(* PLC project HydMotion Functions library, Porcheson AuxBAse Framework 0.0 *)
(* stored: creationDateTime 2023-02-10T00:00:00, modificationDateTime 2026-02-10T00:00:00 *)

TYPE HDY_AxisMotion : STRUCT
  SEGMENTTAG : USINT;
  PLANNER : USINT;
  MODE : USINT;
  ENDCONDITION : USINT;
  DIRECTION : USINT;
  SETPOSITION : REAL;
  SETVELOCITY : REAL;  (* 仅在速度/流量控制模式下使用，表示目标速度； *)
  SETFLOW : REAL;  (* 仅在速度/流量控制模式下使用，表示目标流量；在位置控制模式下忽略 *)
  SETPRESSURE : REAL;
  ACCELERATION : REAL;
  DECELERATION : REAL;
  DURATION : REAL;
  PRESSURERAMPRATE : REAL;
  ACTPOSITION : REAL;
  ACTVELOCITY : REAL;
  ACTFLOW : REAL;
  ACTPRESSURE : REAL;
  TIMESTAMP : REAL;
END_STRUCT;
END_TYPE

FUNCTION_BLOCK HDY_MoveProfile
  VAR_INPUT
    EXECUTE : BOOL;
    MOTION : HDY_AxisMotion;
    AXISID : SINT;
    BUFFERMODE : INT;
  END_VAR
  VAR_OUTPUT
    ACTIVE : BOOL;
    BUSY : BOOL;
    DONE : BOOL;
    ERROR : BOOL;
    ERRORID : WORD;
  END_VAR
  VAR
    Execute0 : BOOL;
    Done0 : BOOL;
    Active0 : BOOL;
    _PENDING : BOOL;
    _EXEC_ID : WORD;
  END_VAR

 {{ extern void __mcl_cmd_MoveProfile(HDY_MOVEPROFILE *data__);	__mcl_cmd_MoveProfile(data__);	 }}			
END_FUNCTION_BLOCK

FUNCTION_BLOCK HDY_LoadProfile
  VAR_INPUT
    EXECUTE : BOOL;
    AXISID : SINT;
    MOTION : HDY_AxisMotion;
  END_VAR
  VAR_OUTPUT
    BUSY : BOOL;
    DONE : BOOL;
    ERROR : BOOL;
    ERRORID : WORD;
  END_VAR
  VAR
    Execute0 : BOOL;
    Done0 : BOOL;
  END_VAR

						{{ extern void __mcl_cmd_LoadProfile(HDY_LOADPROFILE *data__);	__mcl_cmd_LoadProfile(data__);	 }}	
					
END_FUNCTION_BLOCK

FUNCTION_BLOCK HDY_Stop
  VAR_INPUT
    EXECUTE : BOOL;
    AXISID : SINT;
    DECELERATION : REAL;
  END_VAR
  VAR_OUTPUT
    BUSY : BOOL;
    DONE : BOOL;
    COMMANDABORTED : BOOL;
    ERROR : BOOL;
    ERRORID : WORD;
  END_VAR
  VAR
    Execute0 : BOOL;
    Done0 : BOOL;
    Active0 : BOOL;
    _PENDING : BOOL;
  END_VAR

						{{ extern void __mcl_cmd_Stop(HDY_STOP *data__);	__mcl_cmd_Stop(data__);	 }}	
					
END_FUNCTION_BLOCK

(* This Function Block commands a controlled motion to a specified absolute position. *)
FUNCTION_BLOCK HDY_MoveAbsolute
  VAR_INPUT
    EXECUTE : BOOL;
    AXISID : SINT;
    ContinuousUpdate : BOOL;
    POSITION : REAL;
    VELOCITY : REAL;
    ACCELERATION : REAL;
    DECELERATION : REAL;
    JERK : REAL;
    DIRECTION : SINT;
    BUFFERMODE : INT;
  END_VAR
  VAR_OUTPUT
    DONE : BOOL;
    BUSY : BOOL;
    ACTIVE : BOOL;
    COMMANDABORTED : BOOL;
    ERROR : BOOL;
    ERRORID : WORD;
  END_VAR
  VAR
    EXECUTE0 : BOOL;
    DONE0 : BOOL;
    ACTIVE0 : BOOL;
    _PENDING : BOOL;
    _EXEC_ID : WORD;
  END_VAR

						{{ extern void __mcl_cmd_MoveAbsolute(HDY_MOVEABSOLUTE*); __mcl_cmd_MoveAbsolute(data__); }}	
					
END_FUNCTION_BLOCK

(* This Function Block commands a never ending controlled motion at a specified velocity. *)
FUNCTION_BLOCK HDY_MoveVelocity
  VAR_INPUT
    EXECUTE : BOOL;
    AXISID : SINT;
    CONTINUOUSUPDATE : BOOL;
    VELOCITY : REAL;
    ACCELERATION : REAL;
    DECELERATION : REAL;
    JERK : REAL;
    DIRECTION : SINT;
    BUFFERMODE : INT;
  END_VAR
  VAR_OUTPUT
    INVELOCITY : BOOL;
    BUSY : BOOL;
    ACTIVE : BOOL;
    COMMANDABORTED : BOOL;
    ERROR : BOOL;
    ERRORID : WORD;
  END_VAR
  VAR
    EXECUTE0 : BOOL;
    INVELOCITY0 : BOOL;
    ACTIVE0 : BOOL;
    _PENDING : BOOL;
    _EXEC_ID : WORD;
  END_VAR

{{ extern void __mcl_cmd_MoveVelocity(HDY_MOVEVELOCITY*); __mcl_cmd_MoveVelocity(data__); }} 
END_FUNCTION_BLOCK

(* This Function Block makes the transition from the state ‘ErrorStop’ to ‘Disabled’ by resetting all internal axis-related errors *)
FUNCTION_BLOCK HDY_Reset
  VAR_INPUT
    EXECUTE : BOOL;
    AXISID : SINT;
  END_VAR
  VAR_OUTPUT
    DONE : BOOL;
    BUSY : BOOL;
    ERROR : BOOL;
    ERRORID : WORD;
  END_VAR
  VAR
    EXECUTE0 : BOOL;
    DONE0 : BOOL;
  END_VAR

{{ extern void __mcl_cmd_Reset(HDY_RESET*); __mcl_cmd_Reset(data__); }} 
END_FUNCTION_BLOCK

(* This Function Block commands pressure closed control. *)
FUNCTION_BLOCK HDY_PressureHandle
  VAR_INPUT
    EXECUTE : BOOL;
    AXISID : SINT;
    PRESSURE : REAL;
    PRESSURERAMPRATE : REAL;
    DURATION : REAL;
    BUFFERMODE : INT;
  END_VAR
  VAR_OUTPUT
    INPRESSURE : BOOL;
    BUSY : BOOL;
    ACTIVE : BOOL;
    COMMANDABORTED : BOOL;
    ERROR : BOOL;
    ERRORID : WORD;
  END_VAR
  VAR
    EXECUTE0 : BOOL;
    INPRESSURE0 : BOOL;
    ACTIVE0 : BOOL;
    _PENDING : BOOL;
    _EXEC_ID : WORD;
  END_VAR

{{ extern void __mcl_cmd_PressureHandle(HDY_PRESSUREHANDLE*); __mcl_cmd_PressureHandle(data__); }} 
END_FUNCTION_BLOCK

(* This allocates a simulation Axis, for testing.One axis per instanciated FB. *)
FUNCTION_BLOCK HDY_CreateMotion
  VAR_INPUT
    USE_RECIPE : BOOL := 0;
    FLOW_TO_PUMPSPEED : REAL := 20.0;
    PUMPSPEED_LIMIT : REAL := 1800.0;
    USE_SIMULATION : BOOL := 0;
  END_VAR
  VAR_OUTPUT
    AXISID : SINT;
    BUSY : BOOL;
    DONE : BOOL;
    ERROR : BOOL;
    ERRORID : WORD;
  END_VAR
  VAR
    DONE0 : BOOL;
  END_VAR

						{{ extern void __mcl_cmd_CreateMotion(HDY_CREATEMOTION*); __mcl_cmd_CreateMotion(data__); }} 
					
END_FUNCTION_BLOCK

(* set feedback to motion. *)
FUNCTION_BLOCK HDY_SetAxisFeedback
  VAR_INPUT
    ENABLE : BOOL;
    AXISID : SINT;
    ACT_POSITION : REAL;
    ACT_VELOCITY : REAL;
    ACT_FLOW : REAL;
    ACT_PRESSURE : REAL;
    TIMESTAMP : REAL;
  END_VAR
  VAR_OUTPUT
    BUSY : BOOL;
    DONE : BOOL;
    ERROR : BOOL;
    ERRORID : WORD;
  END_VAR
  VAR
    DONE0 : BOOL;
  END_VAR

						{{ extern void __mcl_cmd_SetAxisFeedback(HDY_SETAXISFEEDBACK*); __mcl_cmd_SetAxisFeedback(data__); }} 
					
END_FUNCTION_BLOCK

(* get only one pump speed command from motion. *)
FUNCTION_BLOCK HDY_GetPumpRequest
  VAR_INPUT
    ENABLE : BOOL;
    STRATEGY : SINT;
  END_VAR
  VAR_OUTPUT
    PUMPSPEED : REAL;
    BUSY : BOOL;
    DONE : BOOL;
    ERROR : BOOL;
    ERRORID : WORD;
  END_VAR
  VAR
    DONE0 : BOOL;
  END_VAR

						{{ extern void __mcl_cmd_GetPumpRequest(HDY_GETPUMPREQUEST*); __mcl_cmd_GetPumpRequest(data__); }} 
					
END_FUNCTION_BLOCK

(* get axis status from motion. *)
FUNCTION_BLOCK HDY_ReadStatus
  VAR_INPUT
    ENABLE : BOOL;
    AXISID : SINT;
  END_VAR
  VAR_OUTPUT
    VALID : BOOL;
    BUSY : BOOL;
    ERROR : BOOL;
    ERRORID : WORD;
    STATE : UINT;
  END_VAR

						{{ extern void __mcl_cmd_ReadStatus(HDY_READSTATUS*); __mcl_cmd_ReadStatus(data__); }} 
					
END_FUNCTION_BLOCK

(* get axis error from motion. *)
FUNCTION_BLOCK HDY_ReadError
  VAR_INPUT
    ENABLE : BOOL;
    AXISID : SINT;
  END_VAR
  VAR_OUTPUT
    VALID : BOOL;
    BUSY : BOOL;
    ERROR : BOOL;
    ERRORID : WORD;
  END_VAR

						{{ extern void __mcl_cmd_ReadError(HDY_READERROR*); __mcl_cmd_ReadError(data__); }} 
					
END_FUNCTION_BLOCK
